% RSLogix 500 project I2P-Job-11 Duncan_Sutton.RSS, saved by version 10.00.00.00 %
PROJECT "ML01A"    % processor: Bul.1763 MicroLogix 1100 Series B %

PROGRAM FILES
  LAD 2   8 rungs

DATA FILES
  O0 OUTPUT  4 elements
  I1 INPUT  6 elements
  S2 STATUS  66 elements
  B3 BINARY  1 elements
  T4 TIMER  1 elements
  C5 COUNTER  1 elements
  R6 CONTROL  1 elements
  N7 INTEGER  1 elements
  F8 FLOAT  1 elements

LADDER 2
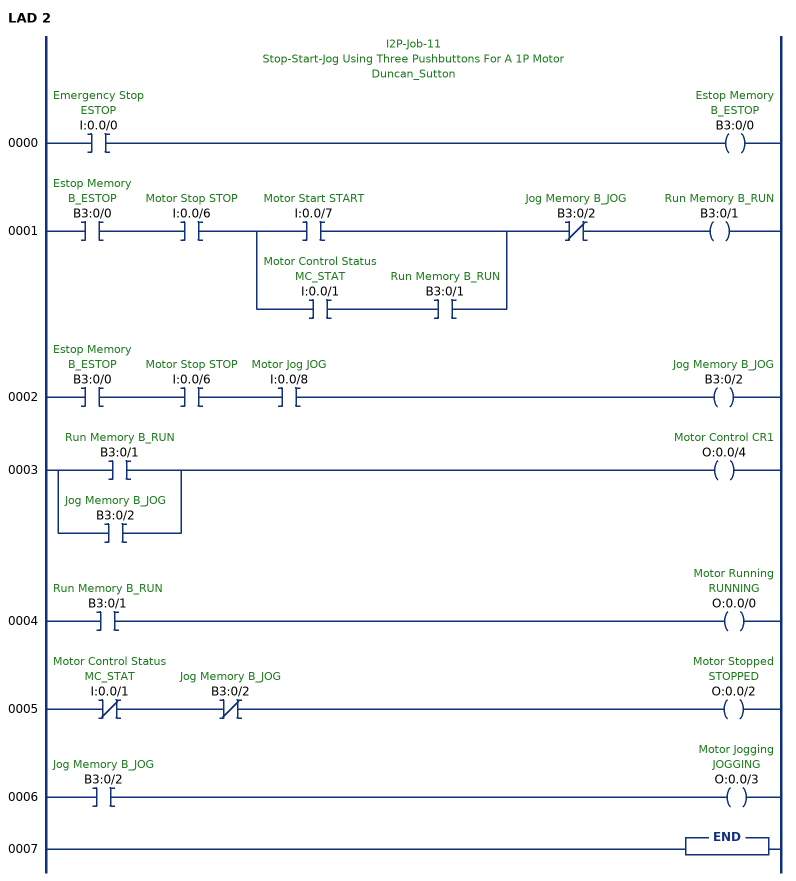
% Rung: 0 %
% I2P-Job-11
% Stop-Start-Jog Using Three Pushbuttons For A 1P Motor
% Duncan_Sutton %
SOR XIC I:0.0/0 OTE B3:0/0 EOR
%   I:0.0/0  ESTOP  "Emergency Stop" %
%   B3:0/0  B_ESTOP  "Estop Memory" %
% Rung: 1 %
SOR XIC B3:0/0 XIC I:0.0/6 BST XIC I:0.0/7 NXB XIC I:0.0/1 XIC B3:0/1 BND XIO B3:0/2 OTE B3:0/1 EOR
%   B3:0/0  B_ESTOP  "Estop Memory" %
%   I:0.0/6  STOP  "Motor Stop" %
%   I:0.0/7  START  "Motor Start" %
%   I:0.0/1  MC_STAT  "Motor Control Status" %
%   B3:0/1  B_RUN  "Run Memory" %
%   B3:0/2  B_JOG  "Jog Memory" %
% Rung: 2 %
SOR XIC B3:0/0 XIC I:0.0/6 XIC I:0.0/8 OTE B3:0/2 EOR
%   B3:0/0  B_ESTOP  "Estop Memory" %
%   I:0.0/6  STOP  "Motor Stop" %
%   I:0.0/8  JOG  "Motor Jog" %
%   B3:0/2  B_JOG  "Jog Memory" %
% Rung: 3 %
SOR BST XIC B3:0/1 NXB XIC B3:0/2 BND OTE O:0.0/4 EOR
%   B3:0/1  B_RUN  "Run Memory" %
%   B3:0/2  B_JOG  "Jog Memory" %
%   O:0.0/4  CR1  "Motor Control" %
% Rung: 4 %
SOR XIC B3:0/1 OTE O:0.0/0 EOR
%   B3:0/1  B_RUN  "Run Memory" %
%   O:0.0/0  RUNNING  "Motor Running" %
% Rung: 5 %
SOR XIO I:0.0/1 XIO B3:0/2 OTE O:0.0/2 EOR
%   I:0.0/1  MC_STAT  "Motor Control Status" %
%   B3:0/2  B_JOG  "Jog Memory" %
%   O:0.0/2  STOPPED  "Motor Stopped" %
% Rung: 6 %
SOR XIC B3:0/2 OTE O:0.0/3 EOR
%   B3:0/2  B_JOG  "Jog Memory" %
%   O:0.0/3  JOGGING  "Motor Jogging" %
% Rung: 7 %
SOR END EOR

OTHER DOCUMENTED ADDRESSES
  I:0.0/2  CR2_C  "Control Relay 2 Contact"
  I:0.0/3  3PSS_PA  "3 Postion Selector Switch Position A"
  I:0.0/4  3PSS_PB  "3 Position Selector Switch Position B"
  I:0.0/5  2PSS_PA  "2 Poistion Selector Switch Position A"
  O:0.0/1  "Yellow Light"
  O:0.0/5  CR_2  "Control Relay 2"
